# EPICS substitutions: modules/event/evrSupport/Db/ioc/IOC-IN20-MC01evr.substitutions
#==============================================================================
#
# Abs:  LCLS EVR IOC records for IN20 MC01
#
# Name: IOC-IN20-MC01evr.substitutions
#
#==============================================================================
#
file evrMCXX.db
{
pattern { DEVICE        }
	{ EVR:IN20:MC01 }
}
